TYPE EL922x_ChannelExtended :
STRUCT
	Status AT%I* : StatusStructExtended;
	Load AT%I* : UINT;
	Current AT%I* : UINT;
	VoltageIn AT%I* : UINT;
	VoltageOut AT%I* : UINT;
	Control AT%q* : OutputStruct;
END_STRUCT
END_TYPE

(* stored: Version 1.1.0.1, ProductVersion 3.1.4024.6
   DUT EL922x_ChannelExtended: Id {c499a2b5-0f9b-439b-a36a-d8ffd80465db} *)
